{attribute 'no_explicit_call' := 'Light is a CLASS and must be accessed using methods or properties'}
FUNCTION_BLOCK Light implements I_OnCommand, I_OffCommand
VAR
	light					AT %Q*: BOOL;
END_VAR


// The body of a class must not be used for code.  
// Cyclic code should be called from a method if needed.

PROPERTY IsOff : BOOL
GET
IsOff := not light;
END_GET
END_PROPERTY

PROPERTY IsOn : BOOL
GET
END_GET
END_PROPERTY

METHOD Off
light := false;
END_METHOD

METHOD On
light := true;
END_METHOD

END_FUNCTION_BLOCK

(* stored: Version 1.1.0.1, ProductVersion 3.1.4024.11
   POU Light: Id {2bb45fa0-3732-4d74-a4f9-b70107719025}, SpecialFunc None
   Property IsOff: Id {78e54d08-811e-4945-b835-8691977f6494}
   Get Get: Id {5da50030-e89d-4dbd-9bf3-7cfbf314ece6}
   Property IsOn: Id {0b89753b-236a-4402-b59b-016dd3f00d33}
   Get Get: Id {a580becd-aae1-45d3-92bd-358e35cdb7c3}
   Method Off: Id {caa3962d-eaab-459a-b06e-1011f201ab27}
   Method On: Id {afa2321b-0383-4b58-9354-3518975e1088} *)
